TYPE DrillingComRequest :
STRUCT
  Start : BOOL;
  Stop : BOOL;
  GoHome : BOOL;
  Halt : BOOL;
END_STRUCT
END_TYPE

(* stored: Version 1.1.0.1
   DUT DrillingComRequest: Id {84109d1b-efca-4afa-9278-03bec9bc4fa3} *)
